% RSLogix 500 project two_way_signal.RSS, saved by version 8.30.00.16 %
PROJECT "UNTITLED"    % processor: Bul.1763 MicroLogix 1100 Series B %

PROGRAM FILES
  LAD 2   5 rungs

DATA FILES
  O0 OUTPUT  4 elements
  I1 INPUT  6 elements
  S2 STATUS  66 elements
  B3 BINARY  1 elements
  T4 TIMER  4 elements
  C5 COUNTER  1 elements
  R6 CONTROL  1 elements
  N7 INTEGER  1 elements
  F8 FLOAT  1 elements

LADDER 2
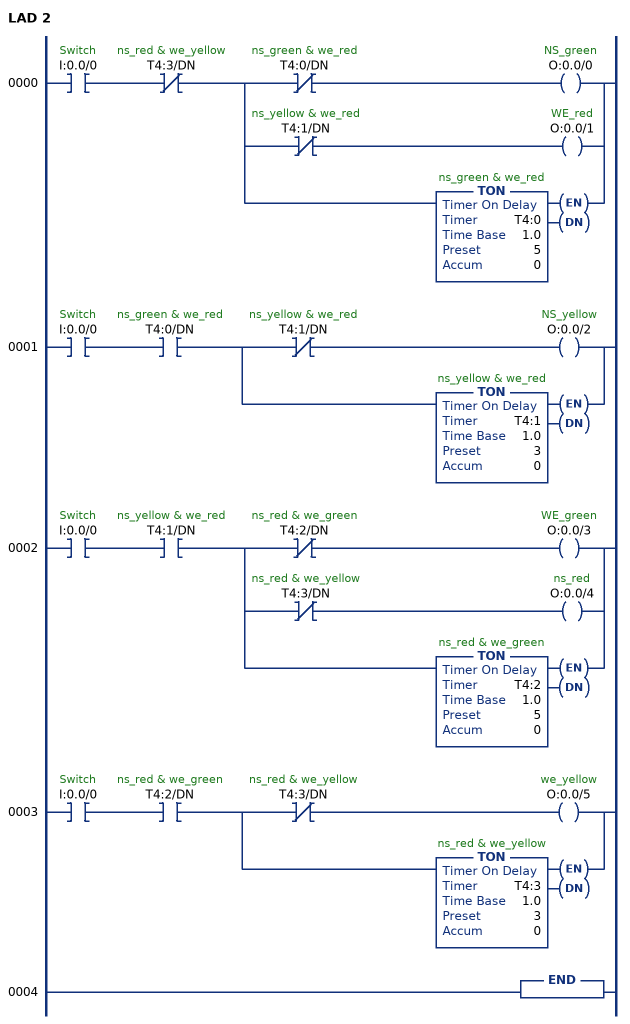
% Rung: 0 %
SOR XIC I:0.0/0 XIO T4:3/DN BST BST XIO T4:0/DN OTE O:0.0/0 NXB XIO T4:1/DN OTE O:0.0/1 BND NXB TON T4:0 1.0 5 0 BND EOR
%   I:0.0/0  "Switch" %
%   T4:3/DN  "ns_red & we_yellow" %
%   T4:0/DN  "ns_green & we_red" %
%   O:0.0/0  "NS_green" %
%   T4:1/DN  "ns_yellow & we_red" %
%   O:0.0/1  "WE_red" %
%   T4:0  "ns_green & we_red" %
% Rung: 1 %
SOR XIC I:0.0/0 XIC T4:0/DN BST XIO T4:1/DN OTE O:0.0/2 NXB TON T4:1 1.0 3 0 BND EOR
%   I:0.0/0  "Switch" %
%   T4:0/DN  "ns_green & we_red" %
%   T4:1/DN  "ns_yellow & we_red" %
%   O:0.0/2  "NS_yellow" %
%   T4:1  "ns_yellow & we_red" %
% Rung: 2 %
SOR XIC I:0.0/0 XIC T4:1/DN BST BST XIO T4:2/DN OTE O:0.0/3 NXB XIO T4:3/DN OTE O:0.0/4 BND NXB TON T4:2 1.0 5 0 BND EOR
%   I:0.0/0  "Switch" %
%   T4:1/DN  "ns_yellow & we_red" %
%   T4:2/DN  "ns_red & we_green" %
%   O:0.0/3  "WE_green" %
%   T4:3/DN  "ns_red & we_yellow" %
%   O:0.0/4  "ns_red" %
%   T4:2  "ns_red & we_green" %
% Rung: 3 %
SOR XIC I:0.0/0 XIC T4:2/DN BST XIO T4:3/DN OTE O:0.0/5 NXB TON T4:3 1.0 3 0 BND EOR
%   I:0.0/0  "Switch" %
%   T4:2/DN  "ns_red & we_green" %
%   T4:3/DN  "ns_red & we_yellow" %
%   O:0.0/5  "we_yellow" %
%   T4:3  "ns_red & we_yellow" %
% Rung: 4 %
SOR END EOR

OTHER DOCUMENTED ADDRESSES
  T4:1.ACC  "ns_yellow & we_red acc"

DATA TABLE (non-zero values as saved)
DATA T4
% .PRE .ACC %
% T4:0 % 5 0
% T4:1 % 3 0
% T4:2 % 5 0
% T4:3 % 3 0
